FUNCTION_BLOCK FB_TestowyPodzespol IMPLEMENTS ITF_StanMaszyny
VAR_INPUT
END_VAR
VAR_OUTPUT
END_VAR
VAR
	bTest: BOOL;
END_VAR

METHOD SM_Aborted : BOOL
END_METHOD

METHOD SM_Aborting : BOOL
END_METHOD

METHOD SM_Clearing : BOOL
END_METHOD

METHOD SM_Complete : BOOL
END_METHOD

METHOD SM_Completing : BOOL
END_METHOD

METHOD SM_Execute : BOOL
END_METHOD

METHOD SM_Held : BOOL
END_METHOD

METHOD SM_Holding : BOOL
END_METHOD

METHOD SM_Idle : BOOL
END_METHOD


METHOD SM_Resetting : BOOL
IF (bTest) THEN
	SM_Resetting							:= TRUE;
ELSE
	SM_Resetting							:= FALSE;
END_IF
END_METHOD

METHOD SM_Starting : BOOL
END_METHOD

METHOD SM_Stopped : BOOL
END_METHOD

METHOD SM_Stopping : BOOL
END_METHOD

METHOD SM_Suspended : BOOL
END_METHOD

METHOD SM_Suspending : BOOL
END_METHOD

METHOD SM_Unholding : BOOL
END_METHOD

METHOD SM_Unsuspending : BOOL
END_METHOD

END_FUNCTION_BLOCK

(* stored: Version 1.1.0.1, ProductVersion 3.1.4024.11
   POU FB_TestowyPodzespol: Id {99f89362-8e9d-468a-b3d0-680272f81d5a}, SpecialFunc None
   Method SM_Aborted: Id {b3adb595-c575-44bc-8e8f-ac910d5547ed}
   Method SM_Aborting: Id {ff86a194-6384-42c7-8a50-5f54004caf4d}
   Method SM_Clearing: Id {9f838446-aca4-43b9-a966-1b05722d56c9}
   Method SM_Complete: Id {56695ff9-28e7-4ca0-a185-779231234124}
   Method SM_Completing: Id {97e9600b-cd0a-40be-bbb7-c741cdbedcef}
   Method SM_Execute: Id {8260b679-a04d-4603-b694-3d98274942b7}
   Method SM_Held: Id {a51677eb-3af3-4e6c-8449-e2965c2a80ac}
   Method SM_Holding: Id {0cc369d8-bbf0-483f-ad05-bc9284a70efd}
   Method SM_Idle: Id {9229ad4d-183a-4ca8-8182-96e655276085}
   Method SM_Resetting: Id {3954a808-3ab2-4ced-8fbe-faa53df131ae}
   Method SM_Starting: Id {5c1e1cdd-7f23-42c7-a2dd-3c86560ba010}
   Method SM_Stopped: Id {2ffa1c49-b6cd-4187-9b87-8703c2b34d01}
   Method SM_Stopping: Id {37127ed8-0483-45a4-8944-3d198debdd83}
   Method SM_Suspended: Id {bb9adbf7-9dea-4619-b3c9-c3933fefc2b8}
   Method SM_Suspending: Id {be6e168b-d458-4148-b196-fd131ff1bd5d}
   Method SM_Unholding: Id {d88c606e-cf74-422c-9d60-f3f4e1d300f4}
   Method SM_Unsuspending: Id {f18588c7-a45d-4239-8fc0-23496702a4c8} *)
